VAR_GLOBAL
	L_EinbruchBild : STRING;
	WetterBild : STRING := BildWolke;
	BildLicht : STRING := GVL_Constants.BildLicht;
END_VAR

(* stored: Version 1.1.0.1, ProductVersion 3.1.4018.5
   GVL Haus4: Id {ca3d3b82-6b66-4ce3-b3c7-182fbb092838} *)
